FUNCTION F_GetColor : DWORD // Return an opaque color in DWORD format for use in visualisation
VAR_INPUT
	Red : BYTE;
	Green : BYTE;
	Blue : BYTE;
END_VAR
VAR
END_VAR

F_GetColor := F_GetTransparantColor(Red, Green, Blue, 16#FF);

END_FUNCTION

(* stored: Version 1.1.0.1, ProductVersion 3.1.4024.11
   POU F_GetColor: Id {d7df149f-d6ac-4a56-9418-435c6968b23b}, SpecialFunc None *)
